FUNCTION_BLOCK OF_E_CYCLE (* Peroidic event generator *)
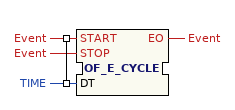
  EVENT_INPUT
    START WITH DT; (* Start the perodic generation of events *)
    STOP; (* Stop the generation of events *)
  END_EVENT
  EVENT_OUTPUT
    EO; (* Periodically triggered output event *)
  END_EVENT
  VAR_INPUT
    DT : TIME; (* cycle time *)
  END_VAR
END_FUNCTION_BLOCK
